{attribute 'qualified_only'}
VAR_GLOBAL
    versionString : STRING := 'v1.2.3';
END_VAR

(* stored: Version 1.1.0.1, ProductVersion 3.1.4024.11
   GVL GVL_Version: Id {178e46eb-caee-44f3-9793-fde14c897d6a} *)
